FUNCTION_BLOCK FB_MCMoveRelative EXTENDS MC_MoveRelative
VAR_INPUT
END_VAR
VAR_OUTPUT
END_VAR
VAR
END_VAR

//FB inherits every funcion from the parent class

END_FUNCTION_BLOCK

(* stored: Version 1.1.0.1, ProductVersion 3.1.4024.12
   POU FB_MCMoveRelative: Id {0eb7de6a-89bd-45de-9b73-ee6b3d62cd32}, SpecialFunc None *)
